FUNCTION_BLOCK FB_CuringStation EXTENDS FB_StepperProgram		// This FB provides an interface for controlling the complete curing station including:
																// Slider and gripper cylinder
																// Temperature control of the heating element
																// Driving of the stepper motor and full control over the 'servo'
																// Camera + lightning
VAR_INPUT
	iGripperOpen:				BOOL;
	iGripperClosed:				BOOL;
	iSliderOpen:				BOOL;
	iSliderClosed:				BOOL;
	iRequestGripperOpen:		BOOL;
	iRequestGripperClosed:		BOOL;
	iRequestSliderOpen:			BOOL;
	iRequestSliderClosed:		BOOL;
	
	iDoStartupTest:				BOOL;
//	iStart:						BOOL;
	
	iEstopOk:					BOOL;	// 1 = System is running, no estop pressed
	iEnable:					BOOL;	// When TRUE, this sequence is possible to be run
	iStationId:					UDINT;	// Station nummer, 1..10
//	iHeatToTestTemp:			BOOL;	// When TRUE, the test program will run 
	iHeatToWorkTemp:			BOOL;	// When TRUE, will start the heating cycle
	iPt100RawValue:				REAL;	// Raw (unscaled value) of the PT100 element (or any other analog input)
	
	iDetectCoupler:				BOOL;
	iDetectMirror:				BOOL;
END_VAR
VAR_OUTPUT
	oGripperToOpen:				BOOL;
	oGripperToClosed:			BOOL;
	oSliderToOpen:				BOOL;
	oSliderToClosed:			BOOL;
	oUnderLightOn:				BOOL;
	oLaserLightOn:				BOOL;
	
	oStartupTestDone:			BOOL;
	oStartupTestFailed:			BOOL;
	oOperational:				BOOL;
	oOperationState:			E_CURING_STATION_OPERATION_STATE;
END_VAR
VAR_IN_OUT
	ioHmi:						ST_CURING_STATION_HMI;
	ioStaticHeaterSettings:		ST_CURING_STATION_HEATER_CONTROL_STATIC_SETTINGS;
END_VAR
VAR
	step:						E_CURING_STATION_SEQUENCE_STEPS;
	service:					ST_CURING_STATION_SERVICE;

	// Devices	
	cyls:						ARRAY[0..1] OF FB_Cylinder;
	heater:						FB_CuringStationHeaterControl;
	//servo:FB_Servo;

	cameraHandler:				FB_CuringStationCameraHandler;
	
	// Helper vars
	gripper:	REFERENCE TO FB_Cylinder;
	slider:		REFERENCE TO FB_Cylinder;
END_VAR
VAR PERSISTENT
	settings:					ST_CURING_STATION_SETTINGS;
END_VAR

IF (NOT IING.cycleStart) THEN
	settings := ioHmi.settings;
END_IF

service := ioHmi.service;

// Helper vars
gripper REF= cyls[0];
slider REF= cyls[1];



callMeRightBeforeSwitchCase(ADR(step));
CASE step OF
	E_CURING_STATION_SEQUENCE_STEPS.INIT:
		gotoNextStep(iDoStartupTest, E_CURING_STATION_SEQUENCE_STEPS.STARTUP_TEST_DO_ECCENTRIC_WHEEL_HOMING);

	E_CURING_STATION_SEQUENCE_STEPS.STARTUP_TEST_DO_ECCENTRIC_WHEEL_HOMING:
		gotoNextStep(TRUE, E_CURING_STATION_SEQUENCE_STEPS.STARTUP_TEST_TEST_SLIDER_TO_WORK);
	
	E_CURING_STATION_SEQUENCE_STEPS.STARTUP_TEST_TEST_SLIDER_TO_WORK:
		gotoNextStep(slider.oInOpenPos, E_CURING_STATION_SEQUENCE_STEPS.STARTUP_TEST_TEST_SLIDER_TO_HOME);

	E_CURING_STATION_SEQUENCE_STEPS.STARTUP_TEST_TEST_SLIDER_TO_HOME:
		gotoNextStep(slider.oInClosedPos, E_CURING_STATION_SEQUENCE_STEPS.STARTUP_TEST_TEST_GRIPPER_TO_WORK);
	
	E_CURING_STATION_SEQUENCE_STEPS.STARTUP_TEST_TEST_GRIPPER_TO_WORK:
		gotoNextStep(gripper.oInOpenPos, E_CURING_STATION_SEQUENCE_STEPS.STARTUP_TEST_TEST_GRIPPER_TO_HOME);

	E_CURING_STATION_SEQUENCE_STEPS.STARTUP_TEST_TEST_GRIPPER_TO_HOME:
		gotoNextStep(gripper.oInClosedPos, E_CURING_STATION_SEQUENCE_STEPS.STARTUP_TEST_TEST_UNDERLIGHT);
	
	E_CURING_STATION_SEQUENCE_STEPS.STARTUP_TEST_TEST_UNDERLIGHT:
		gotoNextStep(cameraHandler.oUnderLightTestOk, E_CURING_STATION_SEQUENCE_STEPS.STARTUP_TEST_TEST_LASER);
		gotoNextStep(cameraHandler.oUnderLightTestFailed, E_CURING_STATION_SEQUENCE_STEPS.STARTUP_TEST_FAIL);
	
	E_CURING_STATION_SEQUENCE_STEPS.STARTUP_TEST_TEST_LASER:
		gotoNextStep(cameraHandler.oLaserLightTestOk, E_CURING_STATION_SEQUENCE_STEPS.STARTUP_TEST_TEST_HEATER);
		gotoNextStep(cameraHandler.oLaserLightTestFailed, E_CURING_STATION_SEQUENCE_STEPS.STARTUP_TEST_FAIL);
	
	E_CURING_STATION_SEQUENCE_STEPS.STARTUP_TEST_TEST_HEATER:
		gotoNextStep(heater.oTestTemperatureReached, E_CURING_STATION_SEQUENCE_STEPS.STARTUP_TEST_DONE);

	E_CURING_STATION_SEQUENCE_STEPS.STARTUP_TEST_DONE:
		gotoNextStep(NOT iDoStartupTest, E_CURING_STATION_SEQUENCE_STEPS.OPERATIONAL);	

	E_CURING_STATION_SEQUENCE_STEPS.STARTUP_TEST_FAIL:
		gotoNextStep(NOT iDoStartupTest, E_CURING_STATION_SEQUENCE_STEPS.INIT);

	E_CURING_STATION_SEQUENCE_STEPS.OPERATIONAL:
		gotoNextStep(iDetectCoupler OR iDetectMirror, E_CURING_STATION_SEQUENCE_STEPS.OPERATIONAL);


ELSE
	step := E_CURING_STATION_SEQUENCE_STEPS.INIT;
END_CASE
callMeRightAfterSwitchCase(TRUE, IING.STRING_BLANK);


slider.iOpenReq := (step = E_CURING_STATION_SEQUENCE_STEPS.STARTUP_TEST_TEST_SLIDER_TO_WORK);
slider.iCloseReq := NOT slider.iOpenReq;

gripper.iOpenReq := (step = E_CURING_STATION_SEQUENCE_STEPS.STARTUP_TEST_TEST_GRIPPER_TO_WORK);
gripper.iCloseReq := NOT gripper.iOpenReq;

heater.iHeatToTestTemp := (step = E_CURING_STATION_SEQUENCE_STEPS.STARTUP_TEST_TEST_HEATER);


cameraHandler(
	iDoUnderLightTest :=		(step = E_CURING_STATION_SEQUENCE_STEPS.STARTUP_TEST_TEST_UNDERLIGHT),
	iDoLaserTest :=				(step = E_CURING_STATION_SEQUENCE_STEPS.STARTUP_TEST_TEST_LASER),
	iDetectCoupler :=			FALSE,
	iDetectMirror :=			FALSE,
	oUnderlightOn =>			oUnderlightOn,
	oLaserLightOn =>			oLaserLightOn
);



// Outputs
oStartupTestFailed := (step = E_CURING_STATION_SEQUENCE_STEPS.STARTUP_TEST_FAIL);
oStartupTestDone := (step = E_CURING_STATION_SEQUENCE_STEPS.STARTUP_TEST_DONE);
oOperational := (step = E_CURING_STATION_SEQUENCE_STEPS.OPERATIONAL);



IF (step = E_CURING_STATION_SEQUENCE_STEPS.OPERATIONAL) THEN
	oOperationState := E_CURING_STATION_OPERATION_STATE.OPERATIONAL;
ELSIF(step = E_CURING_STATION_SEQUENCE_STEPS.STARTUP_TEST_FAIL) THEN
	oOperationState := E_CURING_STATION_OPERATION_STATE.FAULTED;
END_IF

mDevices();
mHmi();

METHOD PRIVATE mDevices
{warning disable C0371}
IF (NOT __ISVALIDREF (ioHmi)) THEN
	RETURN;
END_IF

cyls[0](
	iOpenPos := iGripperOpen,
	iClosePos := iGripperClosed,
	iOpenInterLock := TRUE,
	iCloseInterlock := TRUE,
	iDeactivate := FALSE,
	iDeviceId := FC_2strConcatSeparator(iSeparator := '_', iStr1 := 'Gripper', iStr2 := iDeviceId),
	iControlSignals := iControlSignals,
	oOpen => oGripperToOpen,
	oClose => oGripperToClosed,
	ioHmi := ioHmi.cyls[0]
);


cyls[1](
	iOpenPos := iSliderOpen,
	iClosePos := iSliderClosed,
	iOpenInterLock := TRUE,
	iCloseInterlock := TRUE,
	iDeactivate := FALSE,
	iDeviceId := FC_2strConcatSeparator(iSeparator := '_', iStr1 := 'Slider', iStr2 := iDeviceId),
	iControlSignals := iControlSignals,
	oOpen => oSliderToOpen,
	oClose => oSliderToClosed,
	ioHmi := ioHmi.cyls[1]
);

heater(
	iEstopOk := iEstopOk,
	iEnable := iEnable,
//	iHeatToTestTemp :=,
	iHeatToWorkTemp := iHeatToWorkTemp,
	iPt100RawValue := iPt100RawValue,
	iControlSignals := iControlSignals,
	iDeviceId := FC_2strConcatSeparator(iSeparator := '_', iStr1 := 'Heater', iStr2 := iDeviceId),
	ioHmi := ioHmi.heater,
	ioStaticSettings := ioStaticHeaterSettings, 
);

{warning restore C0371}
END_METHOD

METHOD PRIVATE mHmi
{warning disable C0371}
IF (NOT __ISVALIDREF (ioHmi)) THEN
	RETURN;
END_IF


ioHmi.state.stationId := iStationId;
ioHmi.state.operationState := oOperationState;


ioHmi.settings := settings;
ioHmi.service := service;

{warning restore C0371}
END_METHOD

METHOD PUBLIC stepAsString : T_SHORT_STR
stepAsString := TO_STRING(step);
END_METHOD

END_FUNCTION_BLOCK

(* stored: Version 1.1.0.1
   POU FB_CuringStation: Id {126ed8b3-7cc9-4443-92c2-3634c2f332e1}, SpecialFunc None
   Method mDevices: Id {cfe8be08-49be-425e-8049-4430db425410}
   Method mHmi: Id {c1c4a4bf-1b08-4931-9088-720e2e94e1a9}
   Method stepAsString: Id {1ba0609e-3c25-44f9-a226-3bb5b5742ca9} *)
